// TwinCAT 3 PLC project TcLogTEST
// ProgramVersion: 3.1.4026.12
// libraries:
//   Tc2_Standard, * (Beckhoff Automation GmbH)
//   Tc2_System, * (Beckhoff Automation GmbH)
//   Tc3_Module, * (Beckhoff Automation GmbH)
//   TcLog, * (Benedikt Geisler)
//   TcUnit, * (www.tcunit.org)
// project tree:
//   / TESTS.TcPOU, PlcTask.TcTTO
// (motion and I/O tree: see PLC project tclog)
// real-time tasks:
//   TASK PlcTask1: cycle T#10ms, priority 21, ADS port 351

CONFIGURATION TcLogTEST
    RESOURCE PLC ON TwinCAT3
        TASK PlcTask(INTERVAL := T#10ms, PRIORITY := 21);
        PROGRAM TESTS WITH PlcTask : TESTS;
    END_RESOURCE
END_CONFIGURATION

// ---- TESTS.TcPOU
PROGRAM TESTS
VAR
  DateTime_TEST : DateTime_TEST;
  HelperFunctions_TEST : ConvertAnyToString_TEST;
  DynamicStringBuffer_TEST : DynamicStringBuffer_TEST;
  TestWrapper : TestWrapper_NET();
END_VAR

TcUnit.RUN();

TestWrapper();

END_PROGRAM
